INTERFACE PUBLIC ResettableStateCommands EXTENDS __System.IQueryInterface

METHOD PUBLIC Reset
END_METHOD

END_INTERFACE

(* stored: Version 1.1.0.1, ProductVersion 3.1.4026.18
   Itf ResettableStateCommands: Id {33993280-e484-0e96-1fb6-1f93b1411915}
   Method Reset: Id {3067b572-2c86-00cd-3d4d-873ad3bf1b86} *)
